TYPE User1DUT :
STRUCT
	Int1:INT:=157;
	Int2:INT:=168;
	Bool1:BOOL:=TRUE;
	InInVar:UserInnerInnerDUT;
	Bool2:BOOL:=TRUE;
	Bool3:BOOL:=FALSE;
END_STRUCT
END_TYPE

(* stored: Version 1.1.0.1, ProductVersion 3.1.4024.6
   DUT User1DUT: Id {42076b59-64d0-4d70-b916-3c04b47dabb3} *)
